Staubli VAL3: ioLinks.pgx

program ioLinks()
begin
  //link sock1 - J204 to sSocket sio
  sioLink(sSocket1,io:sock1)
end
